Fanuc KAREL source: ka00205.KL

PROGRAM KA00205
%STACKSIZE=65535
%PRIORITY=65535
%NOLOCKGROUP
-- UNRESOLVED DECLARATIONS (source type spelling not recovered)
-- SRC : ARRAY[4] OF TYPE_0x0013 (type_u16=0x2013)
-- DST : ARRAY[4] OF TYPE_0x0013 (type_u16=0x2013)
BEGIN
-- UNRESOLVED_PC line 7 opcodes [22 22 1E] marker_code=0
END KA00205
